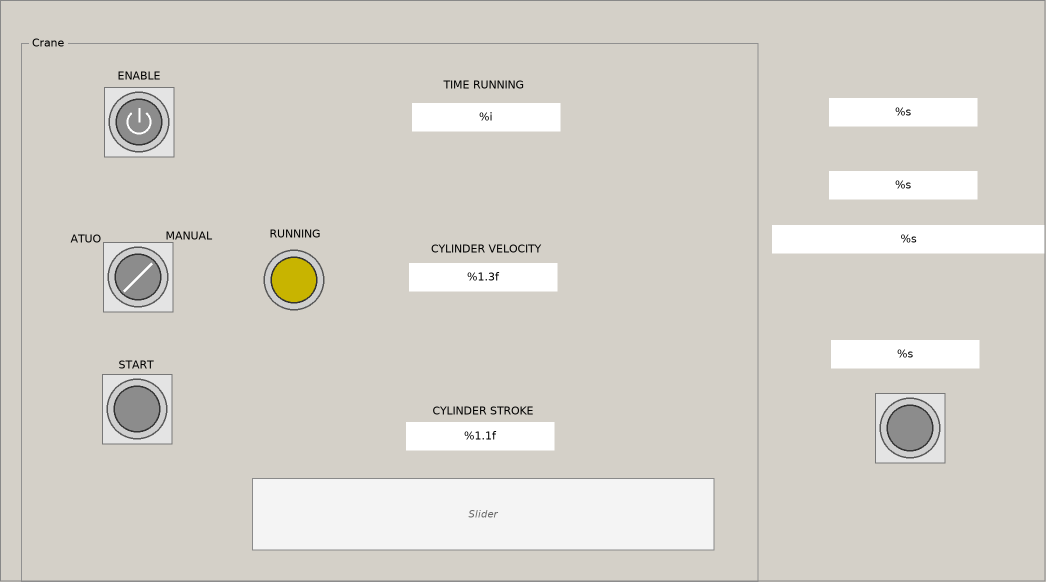
VISUALIZATION CraneHMI  // 1046x582
    Lamp1 (259,245 70x70), variable: output.bRunningLight, style: Lamp-Lamp1-Yellow
    PowerSwitch (104,87 70x70), variable: input.bEnableSwitch, behaviour: TOGGLE, style: Switch-PowerSwitch-Gray
    PushSwitch (102,374 70x70), variable: input.bStartSwitch, behaviour: TOGGLE, style: Switch-PushSwitch-Gray
    RotarySwitch (103,242 70x70), variable: input.bModeSwitch, behaviour: TOGGLE, style: Switch-RotarySwitch-Gray
    Label (114,221 150x30), "MANUAL"
    Label (220,219 150x30), "RUNNING"
    Label (61,350 150x30), "START"
    Label (11,224 150x30), "ATUO"
    Label (64,61 150x30), "ENABLE"
    Textfield (408,262 150x30), "%1.3f", text variable: output.rCylinderVel
    Textfield (405,421 150x30), "%1.1f", text variable: output.rCylinderPos
    Label (411,234 150x30), "CYLINDER VELOCITY"
    Label (408,396 150x30), "CYLINDER STROKE"
    Textfield (411,102 150x30), "%i", text variable: parameter.rRunTime
    Label (409,70 150x30), "TIME RUNNING"
    Slider (252,478 462x72), variable: parameter.rRefCylinderPos, scale 0..1
    GroupBox (21,35 737x547), "Crane"
    Textfield (828,97 150x30), "%s", text variable: MAIN.eStatus
    Textfield (828,170 150x30), "%s", text variable: MAIN.eMode
    Textfield (771,224 275x30), "%s", text variable: MAIN.sEndStopMessage
    Textfield (830,339 150x30), "%s", text variable: input.rSetInputMaxStroke
    PushSwitch (875,393 70x70), variable: input.bSetNewMaxStrokeSwitch, behaviour: TOGGLE, style: Switch-PushSwitch-Gray
END_VISUALIZATION

(* stored: Version 1.1.0.1, ProductVersion 3.1.4024.10
   Visu CraneHMI: Id {7821159e-07b5-4eb8-b327-cf62a5954ee7} *)
